// TIA Portal project "Garage Gate Timer" (V17)
// Garage Gate Timer
// When a car arrives, open the gate for 10 sec. If the car leaves within 1 min, the gate opens automatically.
// After 1 min, the gate will be opened when the status is parking paid.

(* hardware
DEVICE "S7-1200 station_1"  S7-1200 Station
   slot 0: "Rack_0"  S7-1200 Rack  Rack  V1.0
   slot 1: "PLC_1"  CPU 1215C AC/DC/Rly  6ES7 215-1BG40-0XB0  V4.5
*)

// ===== PLC "PLC_1"  CPU 1215C AC/DC/Rly =====

VAR_GLOBAL   // PLC tag table "Default tag table"
   "vehicle_sensor" AT %I0.0 : Bool;
   "gate" AT %Q0.0 : Bool;
   "parking paid" AT %I0.1 : Bool;
   "Tag_1" AT %M0.0 : Bool;
   "Tag_2" AT %M0.1 : Bool;
   "Tag_3" AT %M0.2 : Bool;
END_VAR

// folder: System blocks/Program resources

DATA_BLOCK "IEC_Timer_0_DB"   // DB1
{ S7_Optimized_Access := 'TRUE' }
AUTHOR : Simatic
FAMILY : IEC
NAME : IEC_TMR
VERSION : 1.0
// stored: InstanceOfName IEC_TIMER
"IEC_TIMER"
BEGIN
END_DATA_BLOCK

DATA_BLOCK "IEC_Timer_0_DB_1"   // DB2
{ S7_Optimized_Access := 'TRUE' }
AUTHOR : Simatic
FAMILY : IEC
NAME : IEC_TMR
VERSION : 1.0
// stored: InstanceOfName IEC_TIMER
"IEC_TIMER"
BEGIN
END_DATA_BLOCK

// folder: (top level)

ORGANIZATION_BLOCK "Main"   // OB1, LAD, ProgramCycle
TITLE = "Main Program Sweep (Cycle)"
{ S7_Optimized_Access := 'TRUE' }
VERSION : 0.1
   VAR_INPUT
      Initial_Call : Bool;   // Initial call of this OB
      Remanence : Bool;   // =True, if remanent data are available
   END_VAR
BEGIN

REGION Network 1
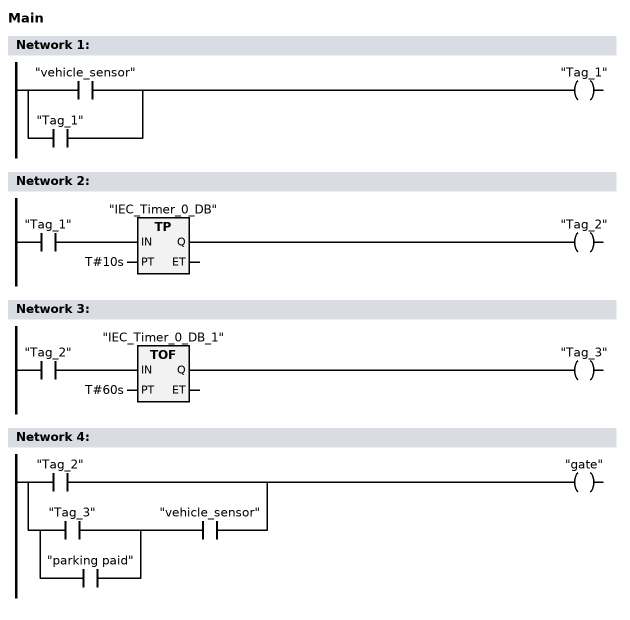
   RUNG wire#powerrail
      Contact( "vehicle_sensor" )
      wire#w1
      Coil( "Tag_1" )
   END_RUNG
   RUNG wire#powerrail
      Contact( "Tag_1" )
   END_RUNG wire#w1
   // the same network as SCL:
   "Tag_1" := "vehicle_sensor" OR "Tag_1";
END_REGION

REGION Network 2
   "IEC_Timer_0_DB".TP(IN := "Tag_1", PT := T#10s);
   "Tag_2" := "IEC_Timer_0_DB".Q;
END_REGION

REGION Network 3
   "IEC_Timer_0_DB_1".TOF(IN := "Tag_2", PT := T#60s);
   "Tag_3" := "IEC_Timer_0_DB_1".Q;
END_REGION

REGION Network 4
   RUNG wire#powerrail
      Contact( "Tag_2" )
      wire#w1
      Coil( "gate" )
   END_RUNG
   RUNG wire#powerrail
      Contact( "Tag_3" )
      wire#w2
      Contact( "vehicle_sensor" )
   END_RUNG wire#w1
   RUNG wire#powerrail
      Contact( "parking paid" )
   END_RUNG wire#w2
   // the same network as SCL:
   "gate" := "Tag_2" OR (("Tag_3" OR "parking paid") AND "vehicle_sensor");
END_REGION
END_ORGANIZATION_BLOCK